TYPE
    ST_ShippingService :
    STRUCT
        AutoMode_ShippingRobot_Left          : REFERENCE TO ST_AutoMode_ShippingRobot_MoveAbs;
        AutoMode_ShippingRobot_Right         : REFERENCE TO ST_AutoMode_ShippingRobot_MoveAbs;
        AutoMode_ShippingRobot_TransmitCVEnd : REFERENCE TO ST_AutoMode_ShippingRobot_MoveAbs;
    END_STRUCT
END_TYPE

(* stored: Version 1.1.0.1, ProductVersion 3.1.4024.13
   DUT ST_ShippingService: Id {0b3c25bc-19ce-45ab-9b06-85beabdcefb6} *)
